// TIA Portal V18 export
// export: Created 2026-06-08T17:01:58.6339435Z, ExportSetting WithDefaults, DisplayName Totally Integrated Automation Portal, DisplayVersion V18, DisplayName TIA Portal Openness, DisplayVersion V18, DisplayName TIA Portal Version Control Interface, DisplayVersion V18, DisplayName STEP 7 Professional, DisplayVersion V18, DisplayName STEP 7 Safety, DisplayVersion V18, DisplayName WinCC Professional, DisplayVersion V18
DATA_BLOCK "M2_I/O_DB"   // DB19
{ S7_Optimized_Access := 'FALSE' }
VERSION : 0.1
// stored: AutoNumber true, DBAccessibleFromOPCUA true, IsOnlyStoredInLoadMemory false, IsWriteProtectedInAS false
   VAR
      RESET_COUNTER : Bool;
      M2_MOVE_R : Bool;
      M2_MOVE_F : Bool;
      M2_STOP : Bool;
   END_VAR
BEGIN
END_DATA_BLOCK
